ABB RobotStudio station: ABB_first_activity_solution.rspag

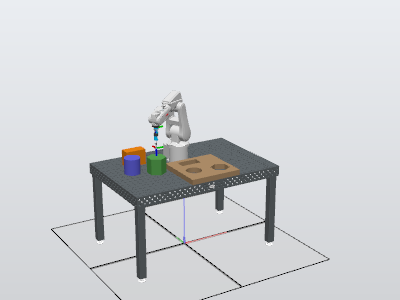
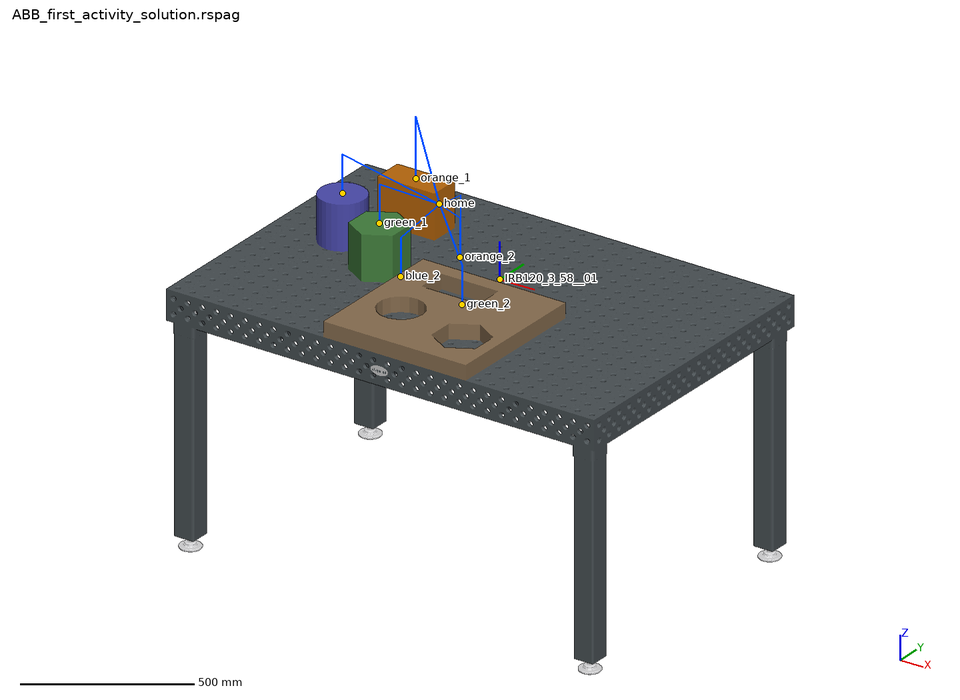
[picture v1: parts stored in the station drawn from their meshes, with robot base, taught points and paths (robot models come from the ABB library and are not in the file)]
--- station ---
Station Solution_1_Tutorial (saved by RobotStudio 22.3.10190.2)
Controller Controller1, task T_ROB1: task frame (RAPID world) sits at (0, 100, 830) mm, rotated rx 0 ry 0 rz -90 deg in the station
Controller Controller1
  mechanical unit ROB_1: IRB120_3_58__01, 6 joints, base frame (0, 0, 0) mm
Layout (positions relative to the parent item):
  - table [part] at (-200, -500, 830) mm, size 500 x 500 x 50 mm
  - object_1 [part] at (-600, -150, 830) mm, size 200 x 100 x 150 mm
  - object_2 [part] at (-650, -150, 830) mm, size 149.5 x 149.7 x 150 mm
  - object_3 [part] at (-700, -200, 830) mm, size 155.5 x 179.5 x 150 mm
  - siegmund_1500_1000 [part], size 1500 x 1010.3 x 830 mm
  - object_11 [part] at (-200, -500, 830) mm, size 200 x 100 x 150 mm
  - object_22 [part] at (-200, -500, 830) mm, size 149.5 x 149.7 x 150 mm
  - object_33 [part] at (-200, -500, 830) mm, size 155.5 x 179.5 x 150 mm
  - IRB120_3_58__01 [mechanism, from Robots\IRB120_3_58_G_01.rslib] at (0, 100, 830) mm, rotated rx 0 ry 0 rz -90 deg; joint values [-1.1286, 0.1686, 0.2297, 0, 1.1726, -1.1286] (rad or m)
  - smc_gripper [mechanism, from Gripper_RS_tool\smc_gripper.rslib] at (-317.07, -50.11, 1261.59) mm, rotated rx 180 ry 0 rz 90 deg
  - Detacher [smart component, from Components\Detacher.rslib]
      properties: Child=object_1; KeepPosition=true
  - Attacher [smart component, from Components\Attacher.rslib]
      properties: Parent=smc_gripper; Flange=0; Child=object_1; Mount=false; Offset=[0 0 0]; Orientation=[0 0 0]
  - Positioner_2 [smart component, from Components\Positioner.rslib]
      properties: Object=object_2; Position=[-0.65 -0.15 0.83]; Orientation=[0 0 0]; Reference=Global; ReferenceObject=(none)
  - Attacher_2 [smart component, from Components\Attacher.rslib]
      properties: Parent=smc_gripper; Flange=0; Child=object_2; Mount=false; Offset=[0 0 0]; Orientation=[0 0 0]
  - Detacher_3 [smart component, from Components\Detacher.rslib]
      properties: Child=object_2; KeepPosition=true
  - Positioner_3 [smart component, from Components\Positioner.rslib]
      properties: Object=object_3; Position=[-0.7 -0.2 0.83]; Orientation=[0 0 0]; Reference=Global; ReferenceObject=(none)
  - Detacher_4 [smart component, from Components\Detacher.rslib]
      properties: Child=object_3; KeepPosition=true
  - Attacher_3 [smart component, from Components\Attacher.rslib]
      properties: Parent=smc_gripper; Flange=0; Child=object_3; Mount=false; Offset=[0 0 0]; Orientation=[0 0 0]
  - Positioner [smart component, from Components\Positioner.rslib]
      properties: Object=object_1; Position=[-0.6 -0.15 0.83]; Orientation=[0 0 0]; Reference=Global; ReferenceObject=(none)
Attachment: smc_gripper is attached to IRB120_3_58__01 / Link6
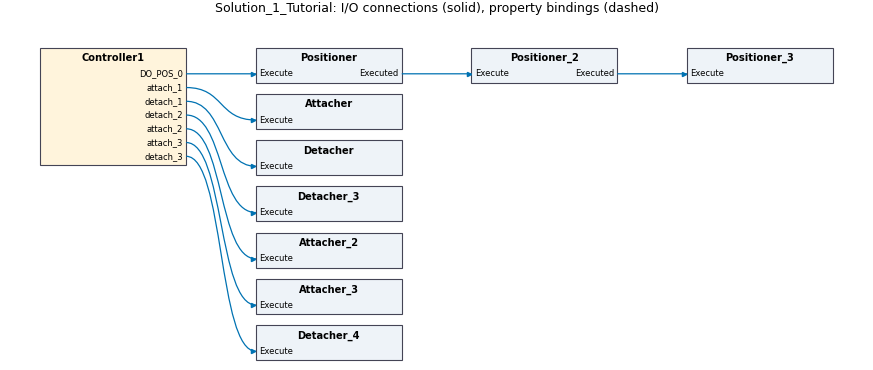
Station logic (signal -> signal, property => property):
  Controller1.DO_POS_0 -> Positioner.Execute
  Controller1.attach_1 -> Attacher.Execute
  Controller1.detach_1 -> Detacher.Execute
  Positioner.Executed -> Positioner_2.Execute
  Controller1.detach_2 -> Detacher_3.Execute
  Controller1.attach_2 -> Attacher_2.Execute
  Positioner_2.Executed -> Positioner_3.Execute
  Controller1.attach_3 -> Attacher_3.Execute
  Controller1.detach_3 -> Detacher_4.Execute
Targets, tools, work objects and paths stored in the station and not in the controller backup, written as RAPID:
! task T_ROB1
MODULE Module1
  PROC Path_10()
    MoveL home,v1000,z100,smc_gripper\WObj:=wobj0;
    MoveL orange_1,v1000,fine,smc_gripper\WObj:=wobj0;
    MoveL orange_2,v1000,fine,smc_gripper\WObj:=wobj0;
  ENDPROC
  PROC Path_20()
    MoveL home,v1000,z100,smc_gripper\WObj:=wobj0;
    MoveL blue_1,v1000,z100,smc_gripper\WObj:=wobj0;
    MoveL blue_2,v1000,z100,smc_gripper\WObj:=wobj0;
  ENDPROC
  PROC Path_30()
    MoveL home,v1000,z100,smc_gripper\WObj:=wobj0;
    MoveL green_1,v1000,z100,smc_gripper\WObj:=wobj0;
    MoveL green_2,v1000,z100,smc_gripper\WObj:=wobj0;
  ENDPROC
ENDMODULE


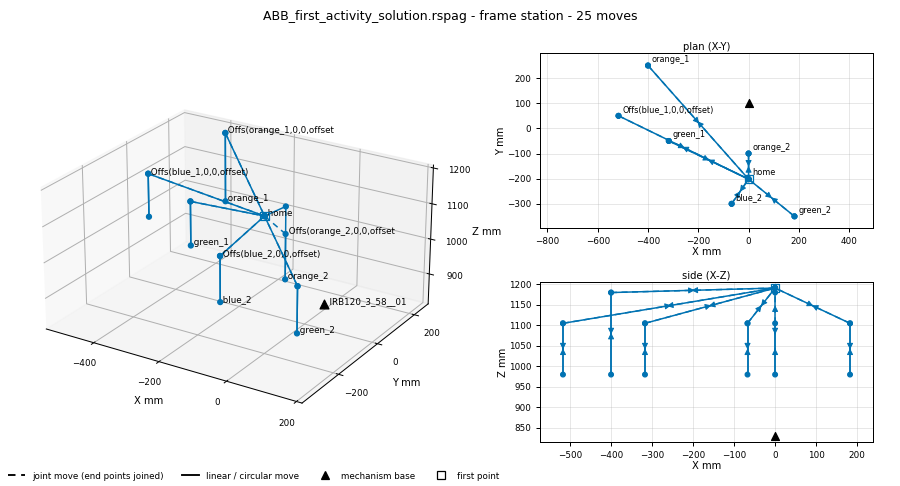
[picture p0: tool path of ABB_first_activity_solution.rspag in frame station, 25 of 25 moves have a stored position in this frame; points joined in program order, loops and branches not executed]
--- Backups/Controller1/RAPID/TASK1/PROGMOD/CalibData.mod ---
MODULE CalibData
    PERS tooldata smc_gripper:=[TRUE,[[0,0.004,197.001],[1,0,0,0]],[1,[0.207,-0.496,71.18],[1,0,0,0],0,0,0]];
ENDMODULE

--- Backups/Controller1/RAPID/TASK1/PROGMOD/Module1.mod ---
MODULE Module1
    CONST robtarget home:=[[301.999956174,0.004,360.999],[-0.000000082,0,1,0],[-1,-1,-1,0],[9E+09,9E+09,9E+09,9E+09,9E+09,9E+09]];
    CONST robtarget orange_1:=[[-150,-400,150],[-0.000000082,0,1,0],[0,0,0,0],[9E+09,9E+09,9E+09,9E+09,9E+09,9E+09]];
    CONST robtarget orange_2:=[[200,0,150],[-0.000000082,0,1,0],[0,0,0,0],[9E+09,9E+09,9E+09,9E+09,9E+09,9E+09]];
    CONST robtarget blue_1:=[[50,-517.298,150.0000082],[-0.000000082,0,1,0],[0,0,0,0],[9E+09,9E+09,9E+09,9E+09,9E+09,9E+09]];
    CONST robtarget blue_2:=[[400,-67.298,150],[-0.000000082,0,1,0],[0,0,0,0],[9E+09,9E+09,9E+09,9E+09,9E+09,9E+09]];
    CONST robtarget green_1:=[[150,-317.298,150],[-0.000000082,0,1,0],[0,0,0,0],[9E+09,9E+09,9E+09,9E+09,9E+09,9E+09]];
    CONST robtarget green_2:=[[450,182.702,150],[-0.000000082,0,1,0],[0,0,0,0],[9E+09,9E+09,9E+09,9E+09,9E+09,9E+09]];

    VAR num offset_orange := 200;
    VAR num offset := 125;


    PROC main()
        PulseDO detach_1;
        PulseDO detach_2;
        PulseDO detach_3;
        PulseDO DO_POS_0;
        MoveJ home,v100,fine,smc_gripper\WObj:=wobj0;

        MoveL Offs(green_1,0,0,offset),v100,z50,smc_gripper\WObj:=wobj0;
        MoveL green_1,v100,fine,smc_gripper\WObj:=wobj0;
        PulseDO attach_3;
        WaitTime 1.0;
        MoveL Offs(green_1,0,0,offset),v100,z50,smc_gripper\WObj:=wobj0;
        MoveJ home,v100,z50,smc_gripper\WObj:=wobj0;
        MoveL Offs(green_2,0,0,offset),v100,z50,smc_gripper\WObj:=wobj0;
        MoveL green_2,v100,fine,smc_gripper\WObj:=wobj0;
        PulseDO detach_3;
        WaitTime 1.0;
        MoveL Offs(green_2,0,0,offset),v100,z50,smc_gripper\WObj:=wobj0;
        MoveJ home,v100,fine,smc_gripper\WObj:=wobj0;
        MoveL Offs(blue_1,0,0,offset),v100,z50,smc_gripper\WObj:=wobj0;
        MoveL [[50,-517.298,150.0000082],[-0.000000082,0,1,0],[0,0,0,0],[9E+09,9E+09,9E+09,9E+09,9E+09,9E+09]],v100,fine,smc_gripper\WObj:=wobj0;
        PulseDO attach_2;
        WaitTime 1.0;
        MoveL Offs(blue_1,0,0,offset),v100,z50,smc_gripper\WObj:=wobj0;
        MoveJ home,v100,z50,smc_gripper\WObj:=wobj0;
        MoveL Offs(blue_2,0,0,offset),v100,z50,smc_gripper\WObj:=wobj0;
        MoveL blue_2,v100,fine,smc_gripper\WObj:=wobj0;
        PulseDO detach_2;
        WaitTime 1.0;
        MoveL Offs(blue_2,0,0,offset),v100,z50,smc_gripper\WObj:=wobj0;
        MoveJ home,v100,fine,smc_gripper\WObj:=wobj0;
        MoveL Offs(orange_1,0,0,offset_orange),v100,z50,smc_gripper\WObj:=wobj0;
        MoveL orange_1,v100,fine,smc_gripper\WObj:=wobj0;
        PulseDO attach_1;
        WaitTime 1.0;
        MoveL Offs(orange_1,0,0,offset_orange),v100,z50,smc_gripper\WObj:=wobj0;
        MoveJ home,v100,z50,smc_gripper\WObj:=wobj0;
        MoveL Offs(orange_2,0,0,offset_orange),v100,z50,smc_gripper\WObj:=wobj0;
        MoveL orange_2,v100,fine,smc_gripper\WObj:=wobj0;
        PulseDO detach_1;
        WaitTime 1.0;
        MoveL Offs(orange_2,0,0,offset),v100,z50,smc_gripper\WObj:=wobj0;
        MoveJ home,v100,fine,smc_gripper\WObj:=wobj0;
    ENDPROC


ENDMODULE

--- Backups/Controller1/SYSPAR/EIO.cfg ---
EIO:CFG_1.0:6:1::
#
EIO_SIGNAL:

      -Name "attach_1" -SignalType "DO"

      -Name "attach_2" -SignalType "DO"

      -Name "attach_3" -SignalType "DO"

      -Name "detach_1" -SignalType "DO"

      -Name "detach_2" -SignalType "DO"

      -Name "detach_3" -SignalType "DO"

      -Name "DO_POS_0" -SignalType "DO"
